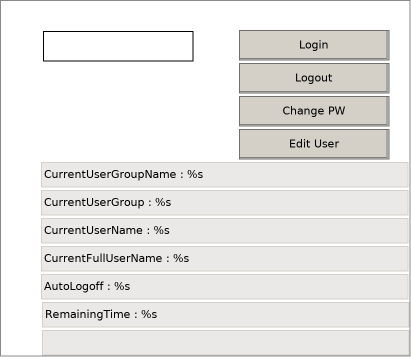
VISUALIZATION Visualization  // 411x357
    Rectangle (43,31 150x30), colour toggle: MAIN.bVar
        OnMouseDown: toggle MAIN.bVar
    Button (239,30 150x30), "Login"
        OnMouseDown: VisuUserMgmt Type=Login
    Button (239,96 150x30), "Change PW"
        OnMouseDown: VisuUserMgmt Type=ChangeUserPassword
    Button (239,129 150x30), "Edit User"
        OnMouseDown: VisuUserMgmt Type=OpenUserConfiguration
    Textfield (41,190 367x25), "CurrentUserGroup : %s", text variable: VisuElems.CurrentUserGroupId
    Textfield (41,218 367x25), "CurrentUserName : %s", text variable: VisuElems.CurrentUserName
    Textfield (41,246 367x25), "CurrentFullUserName : %s", text variable: VisuElems.CurrentFullUserName
    Textfield (41,274 367x25), "AutoLogoff : %s", text variable: VisuElems.CurrentUseAutoLogoutTime
    Textfield (41,162 367x25), "CurrentUserGroupName : %s", text variable: VisuElems.CurrentUserGroupName
    Textfield (42,302 367x25), "RemainingTime : %s", text variable: VisuElems.CurrentRemainingAutoLogoutTime
        OnMouseDown: write the text variable via VisuDialogs.Numpad
    Textfield (42,330 367x25), text list: 'VisuUserMgmt.TL_VUM_Errors', text index: DWORD_TO_STRING(VisuUserManagement.g_udiLastError)
    Button (239,63 150x30), "Logout"
        OnMouseDown: VisuUserMgmt Type=Logout
END_VISUALIZATION

(* stored: Version 1.1.0.1, ProductVersion 3.1.4024.3
   Visu Visualization: Id {291a5a95-1f6c-4d5a-93a2-796520f67c95} *)
